Staubli VAL3: getCycle.pgx

public program getCycle(string& x_sName[], num& x_nTotal[], num& x_nDone[], num x_nIndex, num x_nType)
begin
  // mutex it
  // setMutex
  setMutex(cycleStatus:bMutex)
  // get the cycle from the process LIST
  switch x_nType
    case 0
      if x_nIndex<size(saveCycle:sLoadStart)
        // ON START CYCLE
        x_sName=saveCycle:sLoadStart[x_nIndex]
        x_nTotal=saveCycle:nTotalStart[x_nIndex]
        x_nDone=saveCycle:nDoneStart[x_nIndex]
      endIf
    break
    case 1
      if x_nIndex<size(saveCycle:sLoadProg)
        // get the information about the actual process list
        x_sName=saveCycle:sLoadProg[x_nIndex]
        x_nTotal=saveCycle:nTotalCycle[x_nIndex]
        x_nDone=saveCycle:nDoneCycle[x_nIndex]
      endIf
    break
    case 2
      if x_nIndex<size(saveCycle:sLoadEnd)
        // ON END CYCLE
        x_sName=saveCycle:sLoadEnd[x_nIndex]
        x_nTotal=saveCycle:nTotalEnd[x_nIndex]
        x_nDone=saveCycle:nDoneEnd[x_nIndex]
      endIf
    break
  endSwitch
  // release
  cycleStatus:bMutex=false
end
